REGION Network 25: PART A STATION 2 COLOR STATUS
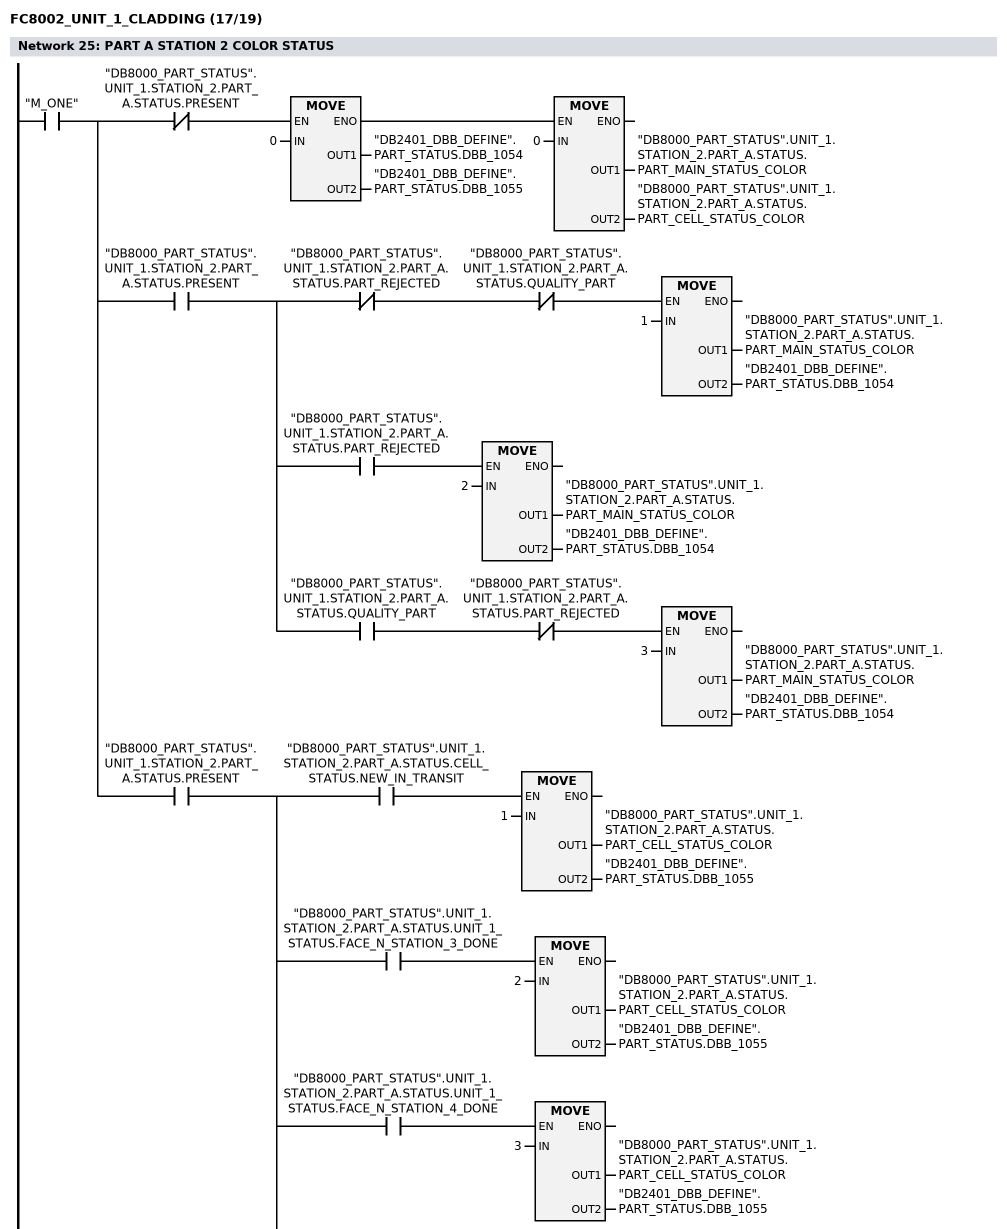
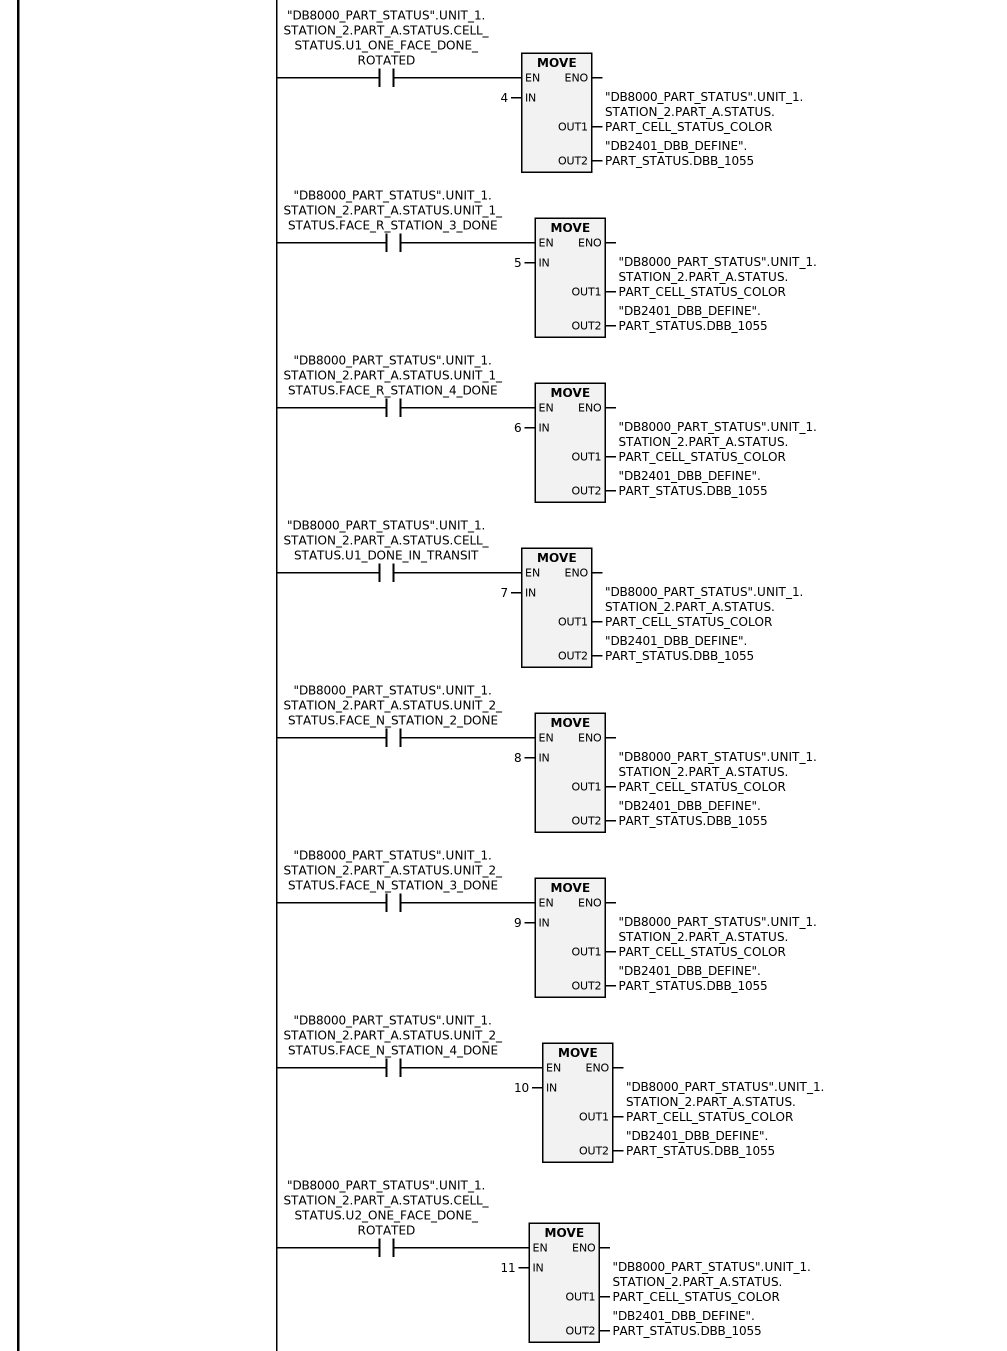
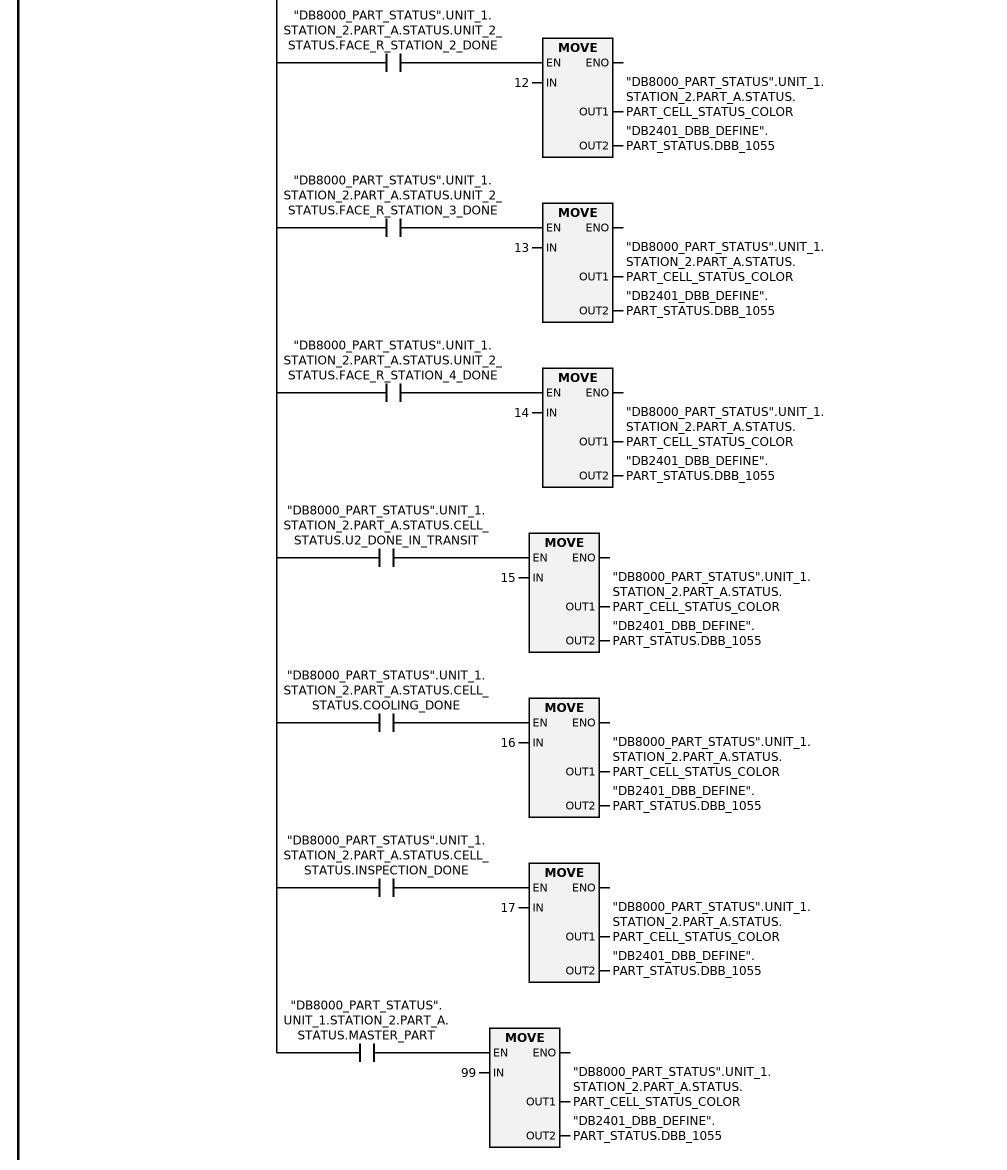
   RUNG wire#powerrail
      Contact( "M_ONE" )
      wire#w1
      I_Contact( "DB8000_PART_STATUS".UNIT_1.STATION_2.PART_A.STATUS.PRESENT )
      { S7_GenerateENO := "TRUE" } Move(in := 0, out1 => "DB2401_DBB_DEFINE".PART_STATUS.DBB_1054, out2 => "DB2401_DBB_DEFINE".PART_STATUS.DBB_1055)
      { S7_GenerateENO := "TRUE" } Move(in := 0, out1 => "DB8000_PART_STATUS".UNIT_1.STATION_2.PART_A.STATUS.PART_MAIN_STATUS_COLOR, out2 => "DB8000_PART_STATUS".UNIT_1.STATION_2.PART_A.STATUS.PART_CELL_STATUS_COLOR)
   END_RUNG
   RUNG wire#w1
      Contact( "DB8000_PART_STATUS".UNIT_1.STATION_2.PART_A.STATUS.PRESENT )
      wire#w2
      I_Contact( "DB8000_PART_STATUS".UNIT_1.STATION_2.PART_A.STATUS.PART_REJECTED )
      I_Contact( "DB8000_PART_STATUS".UNIT_1.STATION_2.PART_A.STATUS.QUALITY_PART )
      { S7_GenerateENO := "TRUE" } Move(in := 1, out1 => "DB8000_PART_STATUS".UNIT_1.STATION_2.PART_A.STATUS.PART_MAIN_STATUS_COLOR, out2 => "DB2401_DBB_DEFINE".PART_STATUS.DBB_1054)
   END_RUNG
   RUNG wire#w2
      Contact( "DB8000_PART_STATUS".UNIT_1.STATION_2.PART_A.STATUS.PART_REJECTED )
      { S7_GenerateENO := "TRUE" } Move(in := 2, out1 => "DB8000_PART_STATUS".UNIT_1.STATION_2.PART_A.STATUS.PART_MAIN_STATUS_COLOR, out2 => "DB2401_DBB_DEFINE".PART_STATUS.DBB_1054)
   END_RUNG
   RUNG wire#w2
      Contact( "DB8000_PART_STATUS".UNIT_1.STATION_2.PART_A.STATUS.QUALITY_PART )
      I_Contact( "DB8000_PART_STATUS".UNIT_1.STATION_2.PART_A.STATUS.PART_REJECTED )
      { S7_GenerateENO := "TRUE" } Move(in := 3, out1 => "DB8000_PART_STATUS".UNIT_1.STATION_2.PART_A.STATUS.PART_MAIN_STATUS_COLOR, out2 => "DB2401_DBB_DEFINE".PART_STATUS.DBB_1054)
   END_RUNG
   RUNG wire#w1
      Contact( "DB8000_PART_STATUS".UNIT_1.STATION_2.PART_A.STATUS.PRESENT )
      wire#w3
      Contact( "DB8000_PART_STATUS".UNIT_1.STATION_2.PART_A.STATUS.CELL_STATUS.NEW_IN_TRANSIT )
      { S7_GenerateENO := "TRUE" } Move(in := 1, out1 => "DB8000_PART_STATUS".UNIT_1.STATION_2.PART_A.STATUS.PART_CELL_STATUS_COLOR, out2 => "DB2401_DBB_DEFINE".PART_STATUS.DBB_1055)
   END_RUNG
   RUNG wire#w3
      Contact( "DB8000_PART_STATUS".UNIT_1.STATION_2.PART_A.STATUS.UNIT_1_STATUS.FACE_N_STATION_3_DONE )
      { S7_GenerateENO := "TRUE" } Move(in := 2, out1 => "DB8000_PART_STATUS".UNIT_1.STATION_2.PART_A.STATUS.PART_CELL_STATUS_COLOR, out2 => "DB2401_DBB_DEFINE".PART_STATUS.DBB_1055)
   END_RUNG
   RUNG wire#w3
      Contact( "DB8000_PART_STATUS".UNIT_1.STATION_2.PART_A.STATUS.UNIT_1_STATUS.FACE_N_STATION_4_DONE )
      { S7_GenerateENO := "TRUE" } Move(in := 3, out1 => "DB8000_PART_STATUS".UNIT_1.STATION_2.PART_A.STATUS.PART_CELL_STATUS_COLOR, out2 => "DB2401_DBB_DEFINE".PART_STATUS.DBB_1055)
   END_RUNG
   RUNG wire#w3
      Contact( "DB8000_PART_STATUS".UNIT_1.STATION_2.PART_A.STATUS.CELL_STATUS.U1_ONE_FACE_DONE_ROTATED )
      { S7_GenerateENO := "TRUE" } Move(in := 4, out1 => "DB8000_PART_STATUS".UNIT_1.STATION_2.PART_A.STATUS.PART_CELL_STATUS_COLOR, out2 => "DB2401_DBB_DEFINE".PART_STATUS.DBB_1055)
   END_RUNG
   RUNG wire#w3
      Contact( "DB8000_PART_STATUS".UNIT_1.STATION_2.PART_A.STATUS.UNIT_1_STATUS.FACE_R_STATION_3_DONE )
      { S7_GenerateENO := "TRUE" } Move(in := 5, out1 => "DB8000_PART_STATUS".UNIT_1.STATION_2.PART_A.STATUS.PART_CELL_STATUS_COLOR, out2 => "DB2401_DBB_DEFINE".PART_STATUS.DBB_1055)
   END_RUNG
   RUNG wire#w3
      Contact( "DB8000_PART_STATUS".UNIT_1.STATION_2.PART_A.STATUS.UNIT_1_STATUS.FACE_R_STATION_4_DONE )
      { S7_GenerateENO := "TRUE" } Move(in := 6, out1 => "DB8000_PART_STATUS".UNIT_1.STATION_2.PART_A.STATUS.PART_CELL_STATUS_COLOR, out2 => "DB2401_DBB_DEFINE".PART_STATUS.DBB_1055)
   END_RUNG
   RUNG wire#w3
      Contact( "DB8000_PART_STATUS".UNIT_1.STATION_2.PART_A.STATUS.CELL_STATUS.U1_DONE_IN_TRANSIT )
      { S7_GenerateENO := "TRUE" } Move(in := 7, out1 => "DB8000_PART_STATUS".UNIT_1.STATION_2.PART_A.STATUS.PART_CELL_STATUS_COLOR, out2 => "DB2401_DBB_DEFINE".PART_STATUS.DBB_1055)
   END_RUNG
   RUNG wire#w3
      Contact( "DB8000_PART_STATUS".UNIT_1.STATION_2.PART_A.STATUS.UNIT_2_STATUS.FACE_N_STATION_2_DONE )
      { S7_GenerateENO := "TRUE" } Move(in := 8, out1 => "DB8000_PART_STATUS".UNIT_1.STATION_2.PART_A.STATUS.PART_CELL_STATUS_COLOR, out2 => "DB2401_DBB_DEFINE".PART_STATUS.DBB_1055)
   END_RUNG
   RUNG wire#w3
      Contact( "DB8000_PART_STATUS".UNIT_1.STATION_2.PART_A.STATUS.UNIT_2_STATUS.FACE_N_STATION_3_DONE )
      Move(in := 9, out1 => "DB8000_PART_STATUS".UNIT_1.STATION_2.PART_A.STATUS.PART_CELL_STATUS_COLOR, out2 => "DB2401_DBB_DEFINE".PART_STATUS.DBB_1055)
   END_RUNG
   RUNG wire#w3
      Contact( "DB8000_PART_STATUS".UNIT_1.STATION_2.PART_A.STATUS.UNIT_2_STATUS.FACE_N_STATION_4_DONE )
      Move(in := 10, out1 => "DB8000_PART_STATUS".UNIT_1.STATION_2.PART_A.STATUS.PART_CELL_STATUS_COLOR, out2 => "DB2401_DBB_DEFINE".PART_STATUS.DBB_1055)
   END_RUNG
   RUNG wire#w3
      Contact( "DB8000_PART_STATUS".UNIT_1.STATION_2.PART_A.STATUS.CELL_STATUS.U2_ONE_FACE_DONE_ROTATED )
      Move(in := 11, out1 => "DB8000_PART_STATUS".UNIT_1.STATION_2.PART_A.STATUS.PART_CELL_STATUS_COLOR, out2 => "DB2401_DBB_DEFINE".PART_STATUS.DBB_1055)
   END_RUNG
   RUNG wire#w3
      Contact( "DB8000_PART_STATUS".UNIT_1.STATION_2.PART_A.STATUS.UNIT_2_STATUS.FACE_R_STATION_2_DONE )
      Move(in := 12, out1 => "DB8000_PART_STATUS".UNIT_1.STATION_2.PART_A.STATUS.PART_CELL_STATUS_COLOR, out2 => "DB2401_DBB_DEFINE".PART_STATUS.DBB_1055)
   END_RUNG
   RUNG wire#w3
      Contact( "DB8000_PART_STATUS".UNIT_1.STATION_2.PART_A.STATUS.UNIT_2_STATUS.FACE_R_STATION_3_DONE )
      Move(in := 13, out1 => "DB8000_PART_STATUS".UNIT_1.STATION_2.PART_A.STATUS.PART_CELL_STATUS_COLOR, out2 => "DB2401_DBB_DEFINE".PART_STATUS.DBB_1055)
   END_RUNG
   RUNG wire#w3
      Contact( "DB8000_PART_STATUS".UNIT_1.STATION_2.PART_A.STATUS.UNIT_2_STATUS.FACE_R_STATION_4_DONE )
      Move(in := 14, out1 => "DB8000_PART_STATUS".UNIT_1.STATION_2.PART_A.STATUS.PART_CELL_STATUS_COLOR, out2 => "DB2401_DBB_DEFINE".PART_STATUS.DBB_1055)
   END_RUNG
   RUNG wire#w3
      Contact( "DB8000_PART_STATUS".UNIT_1.STATION_2.PART_A.STATUS.CELL_STATUS.U2_DONE_IN_TRANSIT )
      Move(in := 15, out1 => "DB8000_PART_STATUS".UNIT_1.STATION_2.PART_A.STATUS.PART_CELL_STATUS_COLOR, out2 => "DB2401_DBB_DEFINE".PART_STATUS.DBB_1055)
   END_RUNG
   RUNG wire#w3
      Contact( "DB8000_PART_STATUS".UNIT_1.STATION_2.PART_A.STATUS.CELL_STATUS.COOLING_DONE )
      Move(in := 16, out1 => "DB8000_PART_STATUS".UNIT_1.STATION_2.PART_A.STATUS.PART_CELL_STATUS_COLOR, out2 => "DB2401_DBB_DEFINE".PART_STATUS.DBB_1055)
   END_RUNG
   RUNG wire#w3
      Contact( "DB8000_PART_STATUS".UNIT_1.STATION_2.PART_A.STATUS.CELL_STATUS.INSPECTION_DONE )
      Move(in := 17, out1 => "DB8000_PART_STATUS".UNIT_1.STATION_2.PART_A.STATUS.PART_CELL_STATUS_COLOR, out2 => "DB2401_DBB_DEFINE".PART_STATUS.DBB_1055)
   END_RUNG
   RUNG wire#w3
      Contact( "DB8000_PART_STATUS".UNIT_1.STATION_2.PART_A.STATUS.MASTER_PART )
      Move(in := 99, out1 => "DB8000_PART_STATUS".UNIT_1.STATION_2.PART_A.STATUS.PART_CELL_STATUS_COLOR, out2 => "DB2401_DBB_DEFINE".PART_STATUS.DBB_1055)
   END_RUNG
   // the same network as SCL:
   // ENO of a box is taken as its EN; it also drops when the box reports an error
   IF "M_ONE" AND NOT "DB8000_PART_STATUS".UNIT_1.STATION_2.PART_A.STATUS.PRESENT THEN
       "DB2401_DBB_DEFINE".PART_STATUS.DBB_1054 := 0;
       "DB2401_DBB_DEFINE".PART_STATUS.DBB_1055 := 0;
       "DB8000_PART_STATUS".UNIT_1.STATION_2.PART_A.STATUS.PART_MAIN_STATUS_COLOR := 0;
       "DB8000_PART_STATUS".UNIT_1.STATION_2.PART_A.STATUS.PART_CELL_STATUS_COLOR := 0;
   END_IF;
   #_w1 := "M_ONE" AND "DB8000_PART_STATUS".UNIT_1.STATION_2.PART_A.STATUS.PRESENT;
   IF #_w1 AND NOT "DB8000_PART_STATUS".UNIT_1.STATION_2.PART_A.STATUS.PART_REJECTED AND NOT "DB8000_PART_STATUS".UNIT_1.STATION_2.PART_A.STATUS.QUALITY_PART THEN
       "DB8000_PART_STATUS".UNIT_1.STATION_2.PART_A.STATUS.PART_MAIN_STATUS_COLOR := 1;
       "DB2401_DBB_DEFINE".PART_STATUS.DBB_1054 := 1;
   END_IF;
   IF #_w1 AND "DB8000_PART_STATUS".UNIT_1.STATION_2.PART_A.STATUS.PART_REJECTED THEN
       "DB8000_PART_STATUS".UNIT_1.STATION_2.PART_A.STATUS.PART_MAIN_STATUS_COLOR := 2;
       "DB2401_DBB_DEFINE".PART_STATUS.DBB_1054 := 2;
   END_IF;
   IF #_w1 AND "DB8000_PART_STATUS".UNIT_1.STATION_2.PART_A.STATUS.QUALITY_PART AND NOT "DB8000_PART_STATUS".UNIT_1.STATION_2.PART_A.STATUS.PART_REJECTED THEN
       "DB8000_PART_STATUS".UNIT_1.STATION_2.PART_A.STATUS.PART_MAIN_STATUS_COLOR := 3;
       "DB2401_DBB_DEFINE".PART_STATUS.DBB_1054 := 3;
   END_IF;
   #_w2 := "M_ONE" AND "DB8000_PART_STATUS".UNIT_1.STATION_2.PART_A.STATUS.PRESENT;
   IF #_w2 AND "DB8000_PART_STATUS".UNIT_1.STATION_2.PART_A.STATUS.CELL_STATUS.NEW_IN_TRANSIT THEN
       "DB8000_PART_STATUS".UNIT_1.STATION_2.PART_A.STATUS.PART_CELL_STATUS_COLOR := 1;
       "DB2401_DBB_DEFINE".PART_STATUS.DBB_1055 := 1;
   END_IF;
   IF #_w2 AND "DB8000_PART_STATUS".UNIT_1.STATION_2.PART_A.STATUS.UNIT_1_STATUS.FACE_N_STATION_3_DONE THEN
       "DB8000_PART_STATUS".UNIT_1.STATION_2.PART_A.STATUS.PART_CELL_STATUS_COLOR := 2;
       "DB2401_DBB_DEFINE".PART_STATUS.DBB_1055 := 2;
   END_IF;
   IF #_w2 AND "DB8000_PART_STATUS".UNIT_1.STATION_2.PART_A.STATUS.UNIT_1_STATUS.FACE_N_STATION_4_DONE THEN
       "DB8000_PART_STATUS".UNIT_1.STATION_2.PART_A.STATUS.PART_CELL_STATUS_COLOR := 3;
       "DB2401_DBB_DEFINE".PART_STATUS.DBB_1055 := 3;
   END_IF;
   IF #_w2 AND "DB8000_PART_STATUS".UNIT_1.STATION_2.PART_A.STATUS.CELL_STATUS.U1_ONE_FACE_DONE_ROTATED THEN
       "DB8000_PART_STATUS".UNIT_1.STATION_2.PART_A.STATUS.PART_CELL_STATUS_COLOR := 4;
       "DB2401_DBB_DEFINE".PART_STATUS.DBB_1055 := 4;
   END_IF;
   IF #_w2 AND "DB8000_PART_STATUS".UNIT_1.STATION_2.PART_A.STATUS.UNIT_1_STATUS.FACE_R_STATION_3_DONE THEN
       "DB8000_PART_STATUS".UNIT_1.STATION_2.PART_A.STATUS.PART_CELL_STATUS_COLOR := 5;
       "DB2401_DBB_DEFINE".PART_STATUS.DBB_1055 := 5;
   END_IF;
   IF #_w2 AND "DB8000_PART_STATUS".UNIT_1.STATION_2.PART_A.STATUS.UNIT_1_STATUS.FACE_R_STATION_4_DONE THEN
       "DB8000_PART_STATUS".UNIT_1.STATION_2.PART_A.STATUS.PART_CELL_STATUS_COLOR := 6;
       "DB2401_DBB_DEFINE".PART_STATUS.DBB_1055 := 6;
   END_IF;
   IF #_w2 AND "DB8000_PART_STATUS".UNIT_1.STATION_2.PART_A.STATUS.CELL_STATUS.U1_DONE_IN_TRANSIT THEN
       "DB8000_PART_STATUS".UNIT_1.STATION_2.PART_A.STATUS.PART_CELL_STATUS_COLOR := 7;
       "DB2401_DBB_DEFINE".PART_STATUS.DBB_1055 := 7;
   END_IF;
   IF #_w2 AND "DB8000_PART_STATUS".UNIT_1.STATION_2.PART_A.STATUS.UNIT_2_STATUS.FACE_N_STATION_2_DONE THEN
       "DB8000_PART_STATUS".UNIT_1.STATION_2.PART_A.STATUS.PART_CELL_STATUS_COLOR := 8;
       "DB2401_DBB_DEFINE".PART_STATUS.DBB_1055 := 8;
   END_IF;
   IF #_w2 AND "DB8000_PART_STATUS".UNIT_1.STATION_2.PART_A.STATUS.UNIT_2_STATUS.FACE_N_STATION_3_DONE THEN
       "DB8000_PART_STATUS".UNIT_1.STATION_2.PART_A.STATUS.PART_CELL_STATUS_COLOR := 9;
       "DB2401_DBB_DEFINE".PART_STATUS.DBB_1055 := 9;
   END_IF;
   IF #_w2 AND "DB8000_PART_STATUS".UNIT_1.STATION_2.PART_A.STATUS.UNIT_2_STATUS.FACE_N_STATION_4_DONE THEN
       "DB8000_PART_STATUS".UNIT_1.STATION_2.PART_A.STATUS.PART_CELL_STATUS_COLOR := 10;
       "DB2401_DBB_DEFINE".PART_STATUS.DBB_1055 := 10;
   END_IF;
   IF #_w2 AND "DB8000_PART_STATUS".UNIT_1.STATION_2.PART_A.STATUS.CELL_STATUS.U2_ONE_FACE_DONE_ROTATED THEN
       "DB8000_PART_STATUS".UNIT_1.STATION_2.PART_A.STATUS.PART_CELL_STATUS_COLOR := 11;
       "DB2401_DBB_DEFINE".PART_STATUS.DBB_1055 := 11;
   END_IF;
   IF #_w2 AND "DB8000_PART_STATUS".UNIT_1.STATION_2.PART_A.STATUS.UNIT_2_STATUS.FACE_R_STATION_2_DONE THEN
       "DB8000_PART_STATUS".UNIT_1.STATION_2.PART_A.STATUS.PART_CELL_STATUS_COLOR := 12;
       "DB2401_DBB_DEFINE".PART_STATUS.DBB_1055 := 12;
   END_IF;
   IF #_w2 AND "DB8000_PART_STATUS".UNIT_1.STATION_2.PART_A.STATUS.UNIT_2_STATUS.FACE_R_STATION_3_DONE THEN
       "DB8000_PART_STATUS".UNIT_1.STATION_2.PART_A.STATUS.PART_CELL_STATUS_COLOR := 13;
       "DB2401_DBB_DEFINE".PART_STATUS.DBB_1055 := 13;
   END_IF;
   IF #_w2 AND "DB8000_PART_STATUS".UNIT_1.STATION_2.PART_A.STATUS.UNIT_2_STATUS.FACE_R_STATION_4_DONE THEN
       "DB8000_PART_STATUS".UNIT_1.STATION_2.PART_A.STATUS.PART_CELL_STATUS_COLOR := 14;
       "DB2401_DBB_DEFINE".PART_STATUS.DBB_1055 := 14;
   END_IF;
   IF #_w2 AND "DB8000_PART_STATUS".UNIT_1.STATION_2.PART_A.STATUS.CELL_STATUS.U2_DONE_IN_TRANSIT THEN
       "DB8000_PART_STATUS".UNIT_1.STATION_2.PART_A.STATUS.PART_CELL_STATUS_COLOR := 15;
       "DB2401_DBB_DEFINE".PART_STATUS.DBB_1055 := 15;
   END_IF;
   IF #_w2 AND "DB8000_PART_STATUS".UNIT_1.STATION_2.PART_A.STATUS.CELL_STATUS.COOLING_DONE THEN
       "DB8000_PART_STATUS".UNIT_1.STATION_2.PART_A.STATUS.PART_CELL_STATUS_COLOR := 16;
       "DB2401_DBB_DEFINE".PART_STATUS.DBB_1055 := 16;
   END_IF;
   IF #_w2 AND "DB8000_PART_STATUS".UNIT_1.STATION_2.PART_A.STATUS.CELL_STATUS.INSPECTION_DONE THEN
       "DB8000_PART_STATUS".UNIT_1.STATION_2.PART_A.STATUS.PART_CELL_STATUS_COLOR := 17;
       "DB2401_DBB_DEFINE".PART_STATUS.DBB_1055 := 17;
   END_IF;
   IF #_w2 AND "DB8000_PART_STATUS".UNIT_1.STATION_2.PART_A.STATUS.MASTER_PART THEN
       "DB8000_PART_STATUS".UNIT_1.STATION_2.PART_A.STATUS.PART_CELL_STATUS_COLOR := 99;
       "DB2401_DBB_DEFINE".PART_STATUS.DBB_1055 := 99;
   END_IF;
END_REGION

REGION Network 26: PART A STATION 3 COLOR STATUS
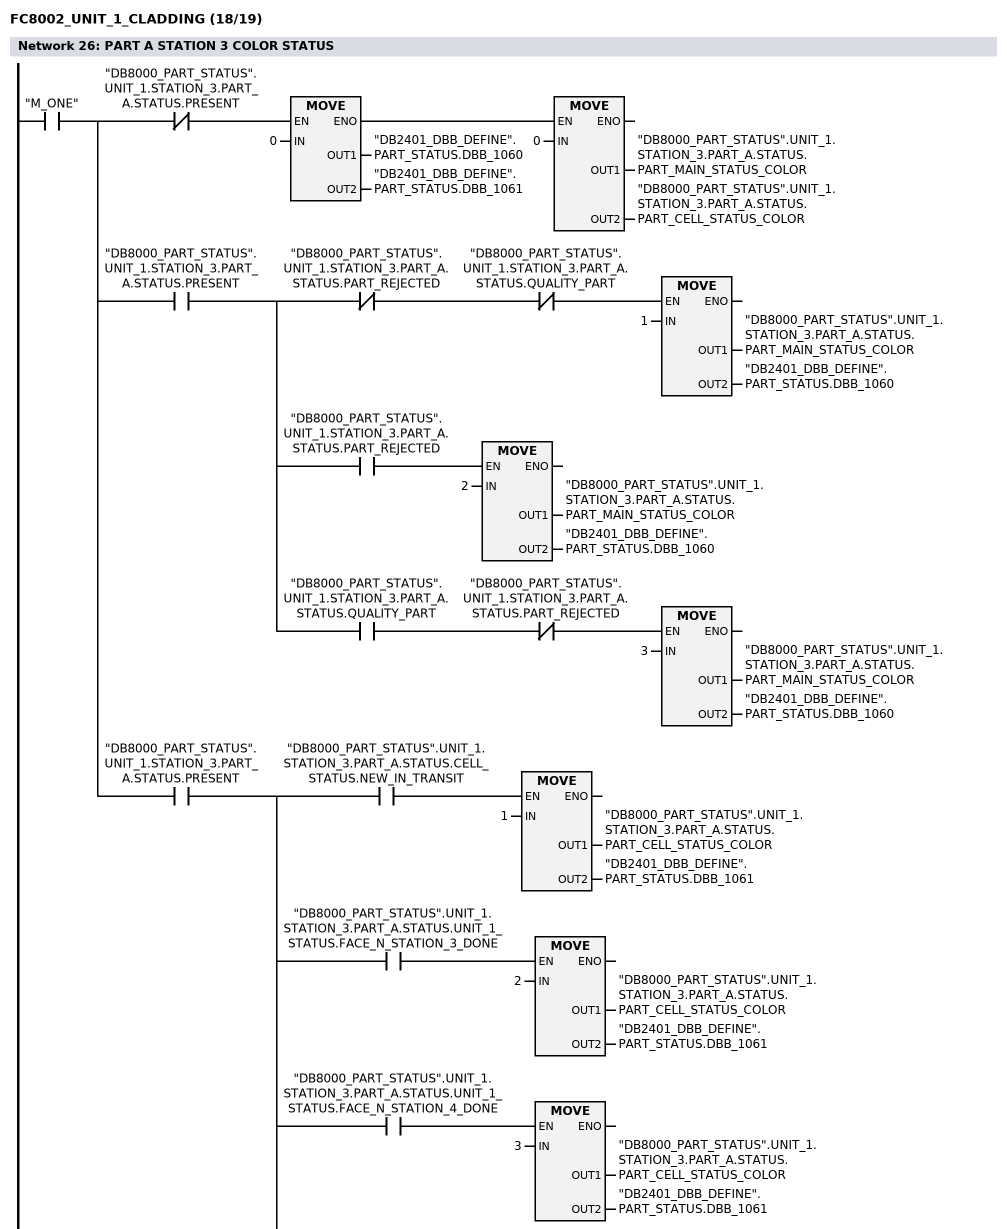
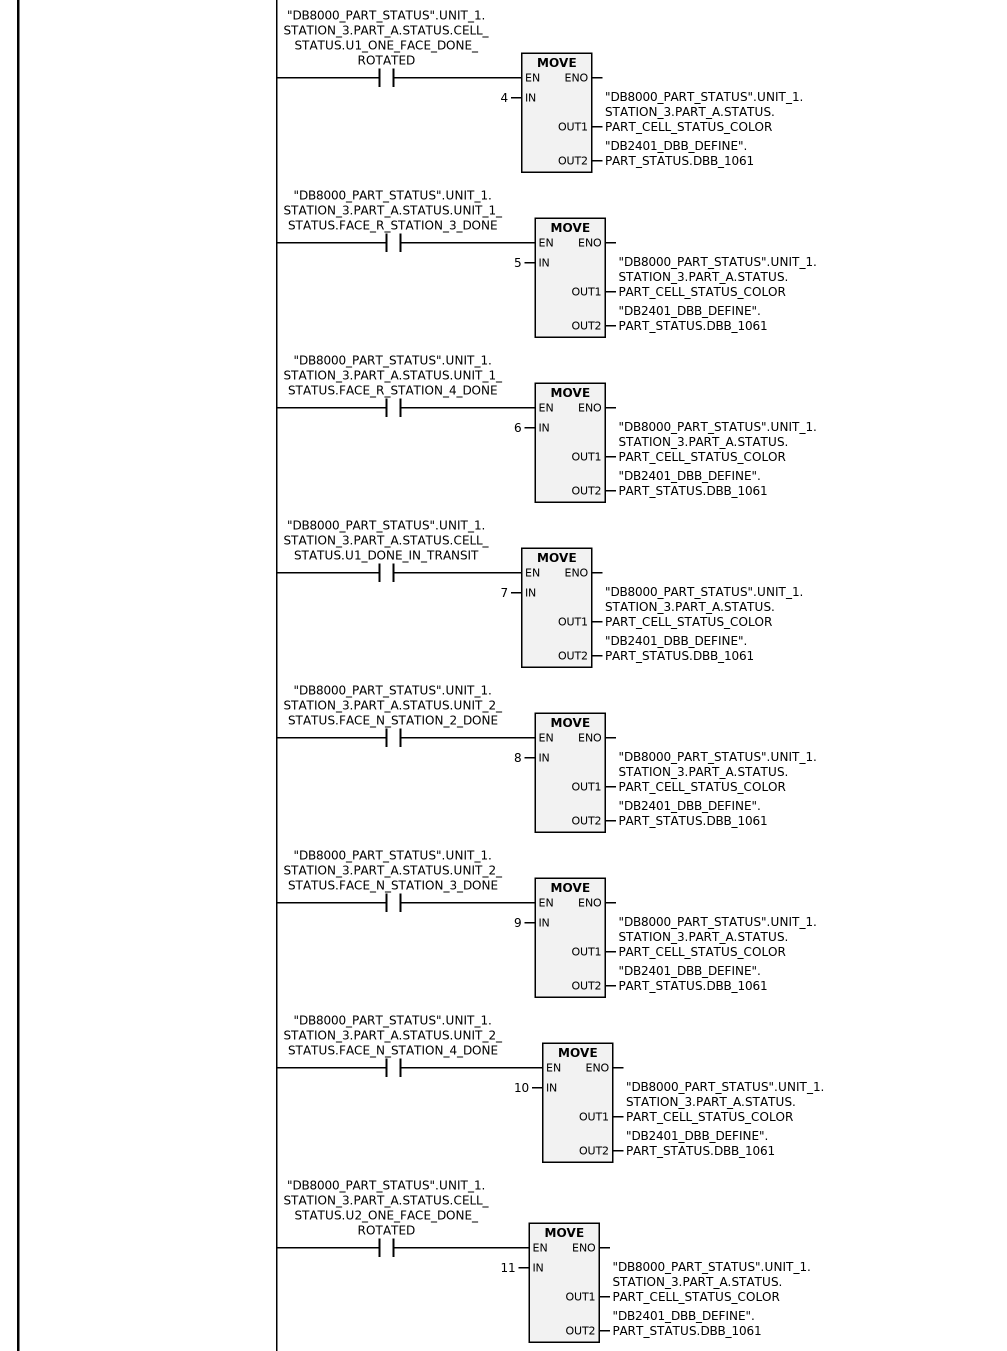
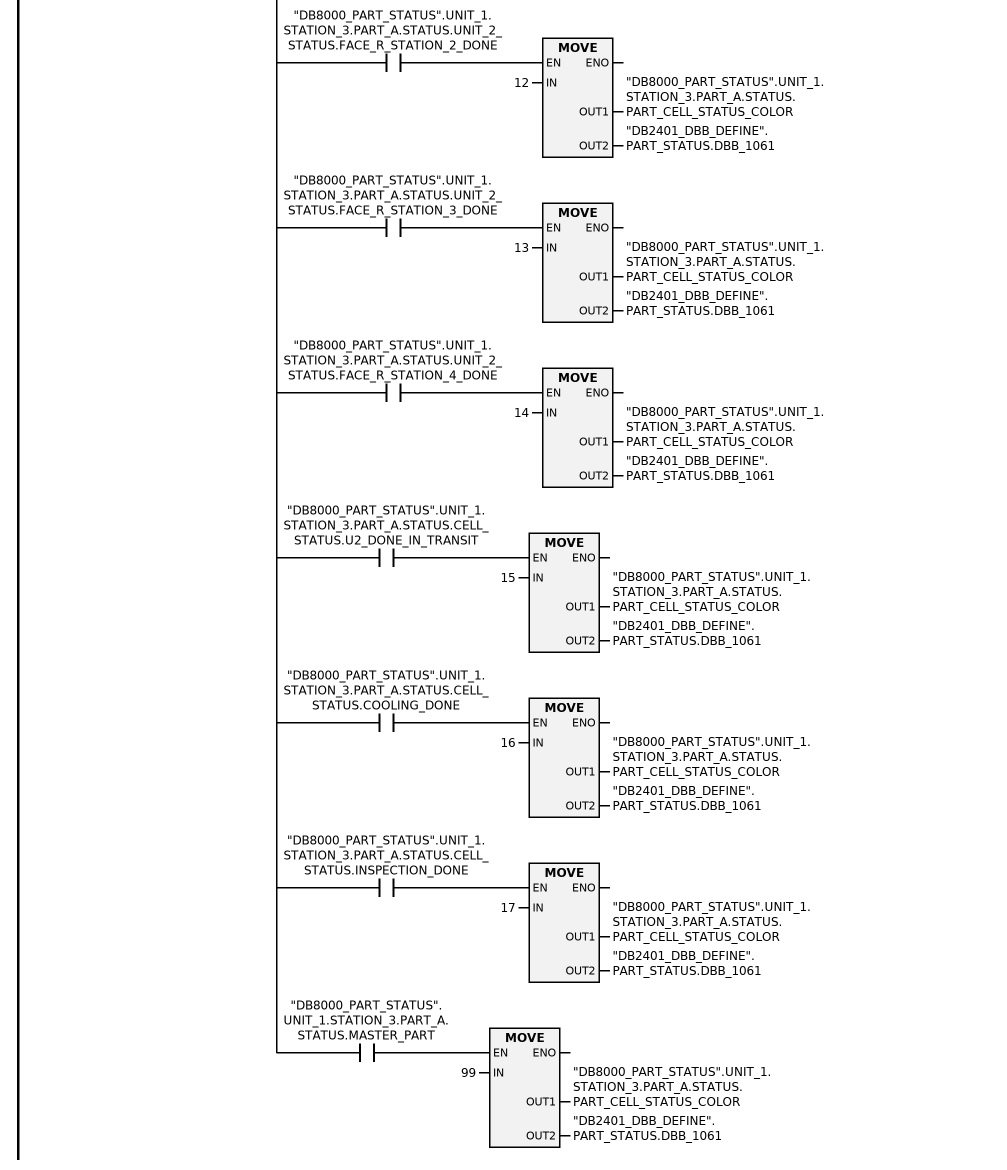
   RUNG wire#powerrail
      Contact( "M_ONE" )
      wire#w1
      I_Contact( "DB8000_PART_STATUS".UNIT_1.STATION_3.PART_A.STATUS.PRESENT )
      { S7_GenerateENO := "TRUE" } Move(in := 0, out1 => "DB2401_DBB_DEFINE".PART_STATUS.DBB_1060, out2 => "DB2401_DBB_DEFINE".PART_STATUS.DBB_1061)
      { S7_GenerateENO := "TRUE" } Move(in := 0, out1 => "DB8000_PART_STATUS".UNIT_1.STATION_3.PART_A.STATUS.PART_MAIN_STATUS_COLOR, out2 => "DB8000_PART_STATUS".UNIT_1.STATION_3.PART_A.STATUS.PART_CELL_STATUS_COLOR)
   END_RUNG
   RUNG wire#w1
      Contact( "DB8000_PART_STATUS".UNIT_1.STATION_3.PART_A.STATUS.PRESENT )
      wire#w2
      I_Contact( "DB8000_PART_STATUS".UNIT_1.STATION_3.PART_A.STATUS.PART_REJECTED )
      I_Contact( "DB8000_PART_STATUS".UNIT_1.STATION_3.PART_A.STATUS.QUALITY_PART )
      { S7_GenerateENO := "TRUE" } Move(in := 1, out1 => "DB8000_PART_STATUS".UNIT_1.STATION_3.PART_A.STATUS.PART_MAIN_STATUS_COLOR, out2 => "DB2401_DBB_DEFINE".PART_STATUS.DBB_1060)
   END_RUNG
   RUNG wire#w2
      Contact( "DB8000_PART_STATUS".UNIT_1.STATION_3.PART_A.STATUS.PART_REJECTED )
      { S7_GenerateENO := "TRUE" } Move(in := 2, out1 => "DB8000_PART_STATUS".UNIT_1.STATION_3.PART_A.STATUS.PART_MAIN_STATUS_COLOR, out2 => "DB2401_DBB_DEFINE".PART_STATUS.DBB_1060)
   END_RUNG
   RUNG wire#w2
      Contact( "DB8000_PART_STATUS".UNIT_1.STATION_3.PART_A.STATUS.QUALITY_PART )
      I_Contact( "DB8000_PART_STATUS".UNIT_1.STATION_3.PART_A.STATUS.PART_REJECTED )
      { S7_GenerateENO := "TRUE" } Move(in := 3, out1 => "DB8000_PART_STATUS".UNIT_1.STATION_3.PART_A.STATUS.PART_MAIN_STATUS_COLOR, out2 => "DB2401_DBB_DEFINE".PART_STATUS.DBB_1060)
   END_RUNG
   RUNG wire#w1
      Contact( "DB8000_PART_STATUS".UNIT_1.STATION_3.PART_A.STATUS.PRESENT )
      wire#w3
      Contact( "DB8000_PART_STATUS".UNIT_1.STATION_3.PART_A.STATUS.CELL_STATUS.NEW_IN_TRANSIT )
      { S7_GenerateENO := "TRUE" } Move(in := 1, out1 => "DB8000_PART_STATUS".UNIT_1.STATION_3.PART_A.STATUS.PART_CELL_STATUS_COLOR, out2 => "DB2401_DBB_DEFINE".PART_STATUS.DBB_1061)
   END_RUNG
   RUNG wire#w3
      Contact( "DB8000_PART_STATUS".UNIT_1.STATION_3.PART_A.STATUS.UNIT_1_STATUS.FACE_N_STATION_3_DONE )
      { S7_GenerateENO := "TRUE" } Move(in := 2, out1 => "DB8000_PART_STATUS".UNIT_1.STATION_3.PART_A.STATUS.PART_CELL_STATUS_COLOR, out2 => "DB2401_DBB_DEFINE".PART_STATUS.DBB_1061)
   END_RUNG
   RUNG wire#w3
      Contact( "DB8000_PART_STATUS".UNIT_1.STATION_3.PART_A.STATUS.UNIT_1_STATUS.FACE_N_STATION_4_DONE )
      { S7_GenerateENO := "TRUE" } Move(in := 3, out1 => "DB8000_PART_STATUS".UNIT_1.STATION_3.PART_A.STATUS.PART_CELL_STATUS_COLOR, out2 => "DB2401_DBB_DEFINE".PART_STATUS.DBB_1061)
   END_RUNG
   RUNG wire#w3
      Contact( "DB8000_PART_STATUS".UNIT_1.STATION_3.PART_A.STATUS.CELL_STATUS.U1_ONE_FACE_DONE_ROTATED )
      { S7_GenerateENO := "TRUE" } Move(in := 4, out1 => "DB8000_PART_STATUS".UNIT_1.STATION_3.PART_A.STATUS.PART_CELL_STATUS_COLOR, out2 => "DB2401_DBB_DEFINE".PART_STATUS.DBB_1061)
   END_RUNG
   RUNG wire#w3
      Contact( "DB8000_PART_STATUS".UNIT_1.STATION_3.PART_A.STATUS.UNIT_1_STATUS.FACE_R_STATION_3_DONE )
      { S7_GenerateENO := "TRUE" } Move(in := 5, out1 => "DB8000_PART_STATUS".UNIT_1.STATION_3.PART_A.STATUS.PART_CELL_STATUS_COLOR, out2 => "DB2401_DBB_DEFINE".PART_STATUS.DBB_1061)
   END_RUNG
   RUNG wire#w3
      Contact( "DB8000_PART_STATUS".UNIT_1.STATION_3.PART_A.STATUS.UNIT_1_STATUS.FACE_R_STATION_4_DONE )
      { S7_GenerateENO := "TRUE" } Move(in := 6, out1 => "DB8000_PART_STATUS".UNIT_1.STATION_3.PART_A.STATUS.PART_CELL_STATUS_COLOR, out2 => "DB2401_DBB_DEFINE".PART_STATUS.DBB_1061)
   END_RUNG
   RUNG wire#w3
      Contact( "DB8000_PART_STATUS".UNIT_1.STATION_3.PART_A.STATUS.CELL_STATUS.U1_DONE_IN_TRANSIT )
      { S7_GenerateENO := "TRUE" } Move(in := 7, out1 => "DB8000_PART_STATUS".UNIT_1.STATION_3.PART_A.STATUS.PART_CELL_STATUS_COLOR, out2 => "DB2401_DBB_DEFINE".PART_STATUS.DBB_1061)
   END_RUNG
   RUNG wire#w3
      Contact( "DB8000_PART_STATUS".UNIT_1.STATION_3.PART_A.STATUS.UNIT_2_STATUS.FACE_N_STATION_2_DONE )
      { S7_GenerateENO := "TRUE" } Move(in := 8, out1 => "DB8000_PART_STATUS".UNIT_1.STATION_3.PART_A.STATUS.PART_CELL_STATUS_COLOR, out2 => "DB2401_DBB_DEFINE".PART_STATUS.DBB_1061)
   END_RUNG
   RUNG wire#w3
      Contact( "DB8000_PART_STATUS".UNIT_1.STATION_3.PART_A.STATUS.UNIT_2_STATUS.FACE_N_STATION_3_DONE )
      Move(in := 9, out1 => "DB8000_PART_STATUS".UNIT_1.STATION_3.PART_A.STATUS.PART_CELL_STATUS_COLOR, out2 => "DB2401_DBB_DEFINE".PART_STATUS.DBB_1061)
   END_RUNG
   RUNG wire#w3
      Contact( "DB8000_PART_STATUS".UNIT_1.STATION_3.PART_A.STATUS.UNIT_2_STATUS.FACE_N_STATION_4_DONE )
      Move(in := 10, out1 => "DB8000_PART_STATUS".UNIT_1.STATION_3.PART_A.STATUS.PART_CELL_STATUS_COLOR, out2 => "DB2401_DBB_DEFINE".PART_STATUS.DBB_1061)
   END_RUNG
   RUNG wire#w3
      Contact( "DB8000_PART_STATUS".UNIT_1.STATION_3.PART_A.STATUS.CELL_STATUS.U2_ONE_FACE_DONE_ROTATED )
      Move(in := 11, out1 => "DB8000_PART_STATUS".UNIT_1.STATION_3.PART_A.STATUS.PART_CELL_STATUS_COLOR, out2 => "DB2401_DBB_DEFINE".PART_STATUS.DBB_1061)
   END_RUNG
   RUNG wire#w3
      Contact( "DB8000_PART_STATUS".UNIT_1.STATION_3.PART_A.STATUS.UNIT_2_STATUS.FACE_R_STATION_2_DONE )
      Move(in := 12, out1 => "DB8000_PART_STATUS".UNIT_1.STATION_3.PART_A.STATUS.PART_CELL_STATUS_COLOR, out2 => "DB2401_DBB_DEFINE".PART_STATUS.DBB_1061)
   END_RUNG
   RUNG wire#w3
      Contact( "DB8000_PART_STATUS".UNIT_1.STATION_3.PART_A.STATUS.UNIT_2_STATUS.FACE_R_STATION_3_DONE )
      Move(in := 13, out1 => "DB8000_PART_STATUS".UNIT_1.STATION_3.PART_A.STATUS.PART_CELL_STATUS_COLOR, out2 => "DB2401_DBB_DEFINE".PART_STATUS.DBB_1061)
   END_RUNG
   RUNG wire#w3
      Contact( "DB8000_PART_STATUS".UNIT_1.STATION_3.PART_A.STATUS.UNIT_2_STATUS.FACE_R_STATION_4_DONE )
      Move(in := 14, out1 => "DB8000_PART_STATUS".UNIT_1.STATION_3.PART_A.STATUS.PART_CELL_STATUS_COLOR, out2 => "DB2401_DBB_DEFINE".PART_STATUS.DBB_1061)
   END_RUNG
   RUNG wire#w3
      Contact( "DB8000_PART_STATUS".UNIT_1.STATION_3.PART_A.STATUS.CELL_STATUS.U2_DONE_IN_TRANSIT )
      Move(in := 15, out1 => "DB8000_PART_STATUS".UNIT_1.STATION_3.PART_A.STATUS.PART_CELL_STATUS_COLOR, out2 => "DB2401_DBB_DEFINE".PART_STATUS.DBB_1061)
   END_RUNG
   RUNG wire#w3
      Contact( "DB8000_PART_STATUS".UNIT_1.STATION_3.PART_A.STATUS.CELL_STATUS.COOLING_DONE )
      Move(in := 16, out1 => "DB8000_PART_STATUS".UNIT_1.STATION_3.PART_A.STATUS.PART_CELL_STATUS_COLOR, out2 => "DB2401_DBB_DEFINE".PART_STATUS.DBB_1061)
   END_RUNG
   RUNG wire#w3
      Contact( "DB8000_PART_STATUS".UNIT_1.STATION_3.PART_A.STATUS.CELL_STATUS.INSPECTION_DONE )
      Move(in := 17, out1 => "DB8000_PART_STATUS".UNIT_1.STATION_3.PART_A.STATUS.PART_CELL_STATUS_COLOR, out2 => "DB2401_DBB_DEFINE".PART_STATUS.DBB_1061)
   END_RUNG
   RUNG wire#w3
      Contact( "DB8000_PART_STATUS".UNIT_1.STATION_3.PART_A.STATUS.MASTER_PART )
      Move(in := 99, out1 => "DB8000_PART_STATUS".UNIT_1.STATION_3.PART_A.STATUS.PART_CELL_STATUS_COLOR, out2 => "DB2401_DBB_DEFINE".PART_STATUS.DBB_1061)
   END_RUNG
   // the same network as SCL:
   // ENO of a box is taken as its EN; it also drops when the box reports an error
   IF "M_ONE" AND NOT "DB8000_PART_STATUS".UNIT_1.STATION_3.PART_A.STATUS.PRESENT THEN
       "DB2401_DBB_DEFINE".PART_STATUS.DBB_1060 := 0;
       "DB2401_DBB_DEFINE".PART_STATUS.DBB_1061 := 0;
       "DB8000_PART_STATUS".UNIT_1.STATION_3.PART_A.STATUS.PART_MAIN_STATUS_COLOR := 0;
       "DB8000_PART_STATUS".UNIT_1.STATION_3.PART_A.STATUS.PART_CELL_STATUS_COLOR := 0;
   END_IF;
   #_w1 := "M_ONE" AND "DB8000_PART_STATUS".UNIT_1.STATION_3.PART_A.STATUS.PRESENT;
   IF #_w1 AND NOT "DB8000_PART_STATUS".UNIT_1.STATION_3.PART_A.STATUS.PART_REJECTED AND NOT "DB8000_PART_STATUS".UNIT_1.STATION_3.PART_A.STATUS.QUALITY_PART THEN
       "DB8000_PART_STATUS".UNIT_1.STATION_3.PART_A.STATUS.PART_MAIN_STATUS_COLOR := 1;
       "DB2401_DBB_DEFINE".PART_STATUS.DBB_1060 := 1;
   END_IF;
   IF #_w1 AND "DB8000_PART_STATUS".UNIT_1.STATION_3.PART_A.STATUS.PART_REJECTED THEN
       "DB8000_PART_STATUS".UNIT_1.STATION_3.PART_A.STATUS.PART_MAIN_STATUS_COLOR := 2;
       "DB2401_DBB_DEFINE".PART_STATUS.DBB_1060 := 2;
   END_IF;
   IF #_w1 AND "DB8000_PART_STATUS".UNIT_1.STATION_3.PART_A.STATUS.QUALITY_PART AND NOT "DB8000_PART_STATUS".UNIT_1.STATION_3.PART_A.STATUS.PART_REJECTED THEN
       "DB8000_PART_STATUS".UNIT_1.STATION_3.PART_A.STATUS.PART_MAIN_STATUS_COLOR := 3;
       "DB2401_DBB_DEFINE".PART_STATUS.DBB_1060 := 3;
   END_IF;
   #_w2 := "M_ONE" AND "DB8000_PART_STATUS".UNIT_1.STATION_3.PART_A.STATUS.PRESENT;
   IF #_w2 AND "DB8000_PART_STATUS".UNIT_1.STATION_3.PART_A.STATUS.CELL_STATUS.NEW_IN_TRANSIT THEN
       "DB8000_PART_STATUS".UNIT_1.STATION_3.PART_A.STATUS.PART_CELL_STATUS_COLOR := 1;
       "DB2401_DBB_DEFINE".PART_STATUS.DBB_1061 := 1;
   END_IF;
   IF #_w2 AND "DB8000_PART_STATUS".UNIT_1.STATION_3.PART_A.STATUS.UNIT_1_STATUS.FACE_N_STATION_3_DONE THEN
       "DB8000_PART_STATUS".UNIT_1.STATION_3.PART_A.STATUS.PART_CELL_STATUS_COLOR := 2;
       "DB2401_DBB_DEFINE".PART_STATUS.DBB_1061 := 2;
   END_IF;
   IF #_w2 AND "DB8000_PART_STATUS".UNIT_1.STATION_3.PART_A.STATUS.UNIT_1_STATUS.FACE_N_STATION_4_DONE THEN
       "DB8000_PART_STATUS".UNIT_1.STATION_3.PART_A.STATUS.PART_CELL_STATUS_COLOR := 3;
       "DB2401_DBB_DEFINE".PART_STATUS.DBB_1061 := 3;
   END_IF;
   IF #_w2 AND "DB8000_PART_STATUS".UNIT_1.STATION_3.PART_A.STATUS.CELL_STATUS.U1_ONE_FACE_DONE_ROTATED THEN
       "DB8000_PART_STATUS".UNIT_1.STATION_3.PART_A.STATUS.PART_CELL_STATUS_COLOR := 4;
       "DB2401_DBB_DEFINE".PART_STATUS.DBB_1061 := 4;
   END_IF;
   IF #_w2 AND "DB8000_PART_STATUS".UNIT_1.STATION_3.PART_A.STATUS.UNIT_1_STATUS.FACE_R_STATION_3_DONE THEN
       "DB8000_PART_STATUS".UNIT_1.STATION_3.PART_A.STATUS.PART_CELL_STATUS_COLOR := 5;
       "DB2401_DBB_DEFINE".PART_STATUS.DBB_1061 := 5;
   END_IF;
   IF #_w2 AND "DB8000_PART_STATUS".UNIT_1.STATION_3.PART_A.STATUS.UNIT_1_STATUS.FACE_R_STATION_4_DONE THEN
       "DB8000_PART_STATUS".UNIT_1.STATION_3.PART_A.STATUS.PART_CELL_STATUS_COLOR := 6;
       "DB2401_DBB_DEFINE".PART_STATUS.DBB_1061 := 6;
   END_IF;
   IF #_w2 AND "DB8000_PART_STATUS".UNIT_1.STATION_3.PART_A.STATUS.CELL_STATUS.U1_DONE_IN_TRANSIT THEN
       "DB8000_PART_STATUS".UNIT_1.STATION_3.PART_A.STATUS.PART_CELL_STATUS_COLOR := 7;
       "DB2401_DBB_DEFINE".PART_STATUS.DBB_1061 := 7;
   END_IF;
   IF #_w2 AND "DB8000_PART_STATUS".UNIT_1.STATION_3.PART_A.STATUS.UNIT_2_STATUS.FACE_N_STATION_2_DONE THEN
       "DB8000_PART_STATUS".UNIT_1.STATION_3.PART_A.STATUS.PART_CELL_STATUS_COLOR := 8;
       "DB2401_DBB_DEFINE".PART_STATUS.DBB_1061 := 8;
   END_IF;
   IF #_w2 AND "DB8000_PART_STATUS".UNIT_1.STATION_3.PART_A.STATUS.UNIT_2_STATUS.FACE_N_STATION_3_DONE THEN
       "DB8000_PART_STATUS".UNIT_1.STATION_3.PART_A.STATUS.PART_CELL_STATUS_COLOR := 9;
       "DB2401_DBB_DEFINE".PART_STATUS.DBB_1061 := 9;
   END_IF;
   IF #_w2 AND "DB8000_PART_STATUS".UNIT_1.STATION_3.PART_A.STATUS.UNIT_2_STATUS.FACE_N_STATION_4_DONE THEN
       "DB8000_PART_STATUS".UNIT_1.STATION_3.PART_A.STATUS.PART_CELL_STATUS_COLOR := 10;
       "DB2401_DBB_DEFINE".PART_STATUS.DBB_1061 := 10;
   END_IF;
   IF #_w2 AND "DB8000_PART_STATUS".UNIT_1.STATION_3.PART_A.STATUS.CELL_STATUS.U2_ONE_FACE_DONE_ROTATED THEN
       "DB8000_PART_STATUS".UNIT_1.STATION_3.PART_A.STATUS.PART_CELL_STATUS_COLOR := 11;
       "DB2401_DBB_DEFINE".PART_STATUS.DBB_1061 := 11;
   END_IF;
   IF #_w2 AND "DB8000_PART_STATUS".UNIT_1.STATION_3.PART_A.STATUS.UNIT_2_STATUS.FACE_R_STATION_2_DONE THEN
       "DB8000_PART_STATUS".UNIT_1.STATION_3.PART_A.STATUS.PART_CELL_STATUS_COLOR := 12;
       "DB2401_DBB_DEFINE".PART_STATUS.DBB_1061 := 12;
   END_IF;
   IF #_w2 AND "DB8000_PART_STATUS".UNIT_1.STATION_3.PART_A.STATUS.UNIT_2_STATUS.FACE_R_STATION_3_DONE THEN
       "DB8000_PART_STATUS".UNIT_1.STATION_3.PART_A.STATUS.PART_CELL_STATUS_COLOR := 13;
       "DB2401_DBB_DEFINE".PART_STATUS.DBB_1061 := 13;
   END_IF;
   IF #_w2 AND "DB8000_PART_STATUS".UNIT_1.STATION_3.PART_A.STATUS.UNIT_2_STATUS.FACE_R_STATION_4_DONE THEN
       "DB8000_PART_STATUS".UNIT_1.STATION_3.PART_A.STATUS.PART_CELL_STATUS_COLOR := 14;
       "DB2401_DBB_DEFINE".PART_STATUS.DBB_1061 := 14;
   END_IF;
   IF #_w2 AND "DB8000_PART_STATUS".UNIT_1.STATION_3.PART_A.STATUS.CELL_STATUS.U2_DONE_IN_TRANSIT THEN
       "DB8000_PART_STATUS".UNIT_1.STATION_3.PART_A.STATUS.PART_CELL_STATUS_COLOR := 15;
       "DB2401_DBB_DEFINE".PART_STATUS.DBB_1061 := 15;
   END_IF;
   IF #_w2 AND "DB8000_PART_STATUS".UNIT_1.STATION_3.PART_A.STATUS.CELL_STATUS.COOLING_DONE THEN
       "DB8000_PART_STATUS".UNIT_1.STATION_3.PART_A.STATUS.PART_CELL_STATUS_COLOR := 16;
       "DB2401_DBB_DEFINE".PART_STATUS.DBB_1061 := 16;
   END_IF;
   IF #_w2 AND "DB8000_PART_STATUS".UNIT_1.STATION_3.PART_A.STATUS.CELL_STATUS.INSPECTION_DONE THEN
       "DB8000_PART_STATUS".UNIT_1.STATION_3.PART_A.STATUS.PART_CELL_STATUS_COLOR := 17;
       "DB2401_DBB_DEFINE".PART_STATUS.DBB_1061 := 17;
   END_IF;
   IF #_w2 AND "DB8000_PART_STATUS".UNIT_1.STATION_3.PART_A.STATUS.MASTER_PART THEN
       "DB8000_PART_STATUS".UNIT_1.STATION_3.PART_A.STATUS.PART_CELL_STATUS_COLOR := 99;
       "DB2401_DBB_DEFINE".PART_STATUS.DBB_1061 := 99;
   END_IF;
END_REGION

REGION Network 27: PART A STATION 4 COLOR STATUS
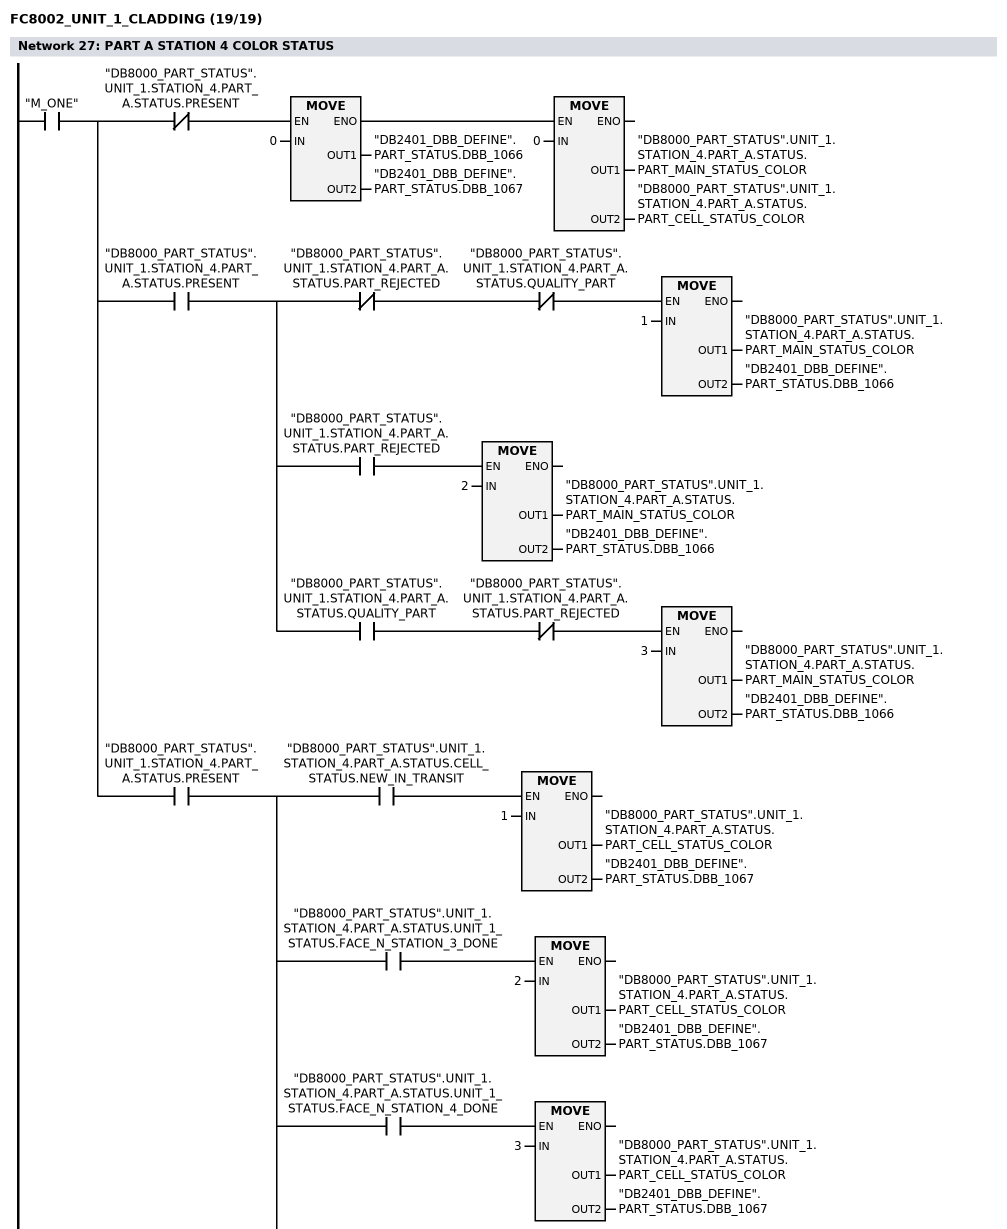
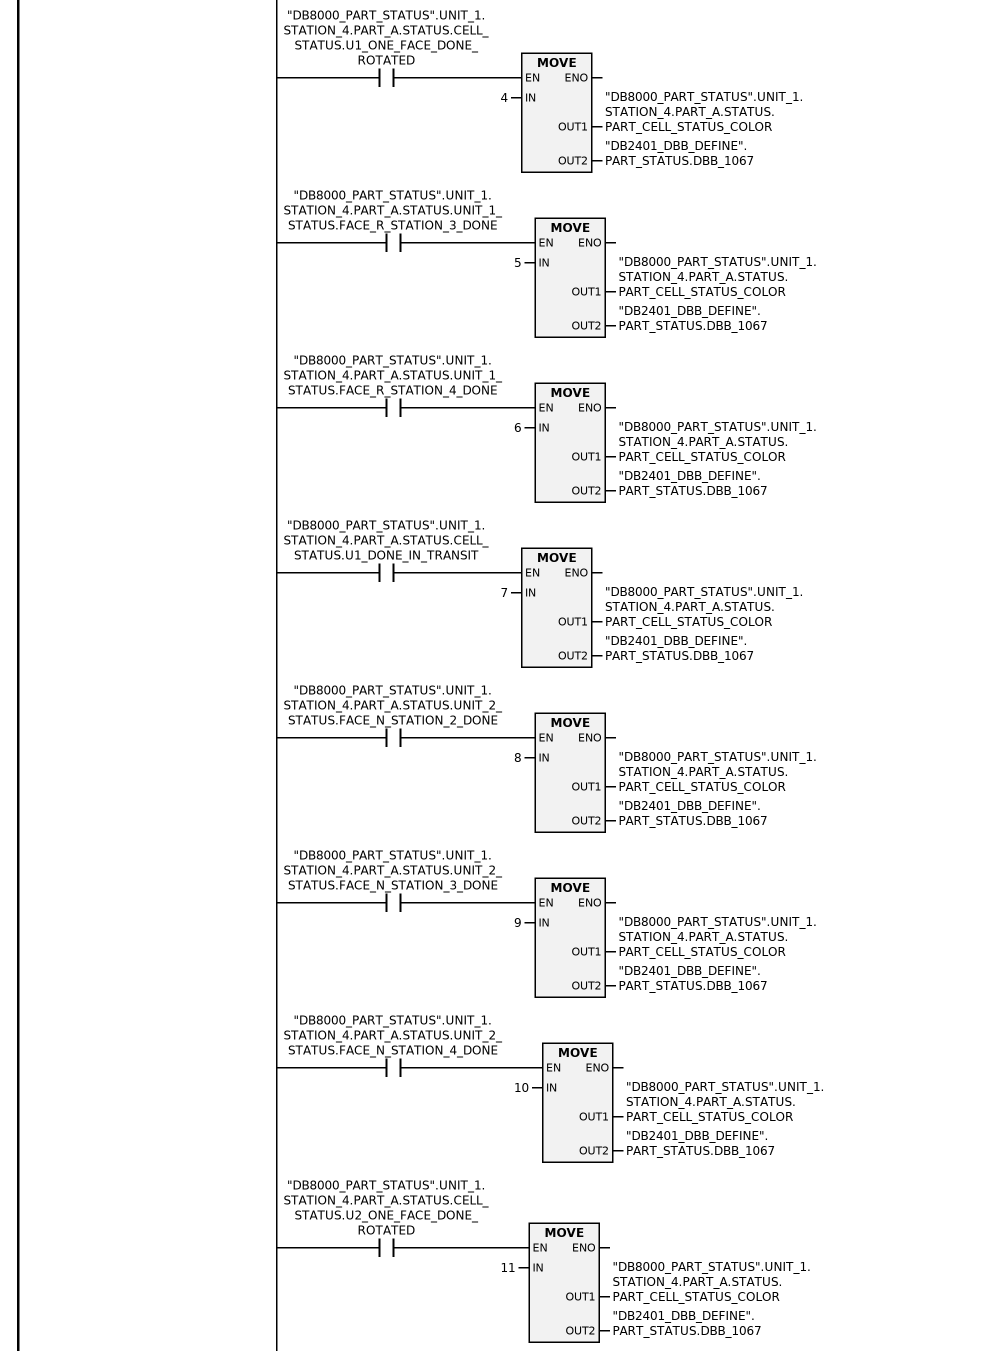
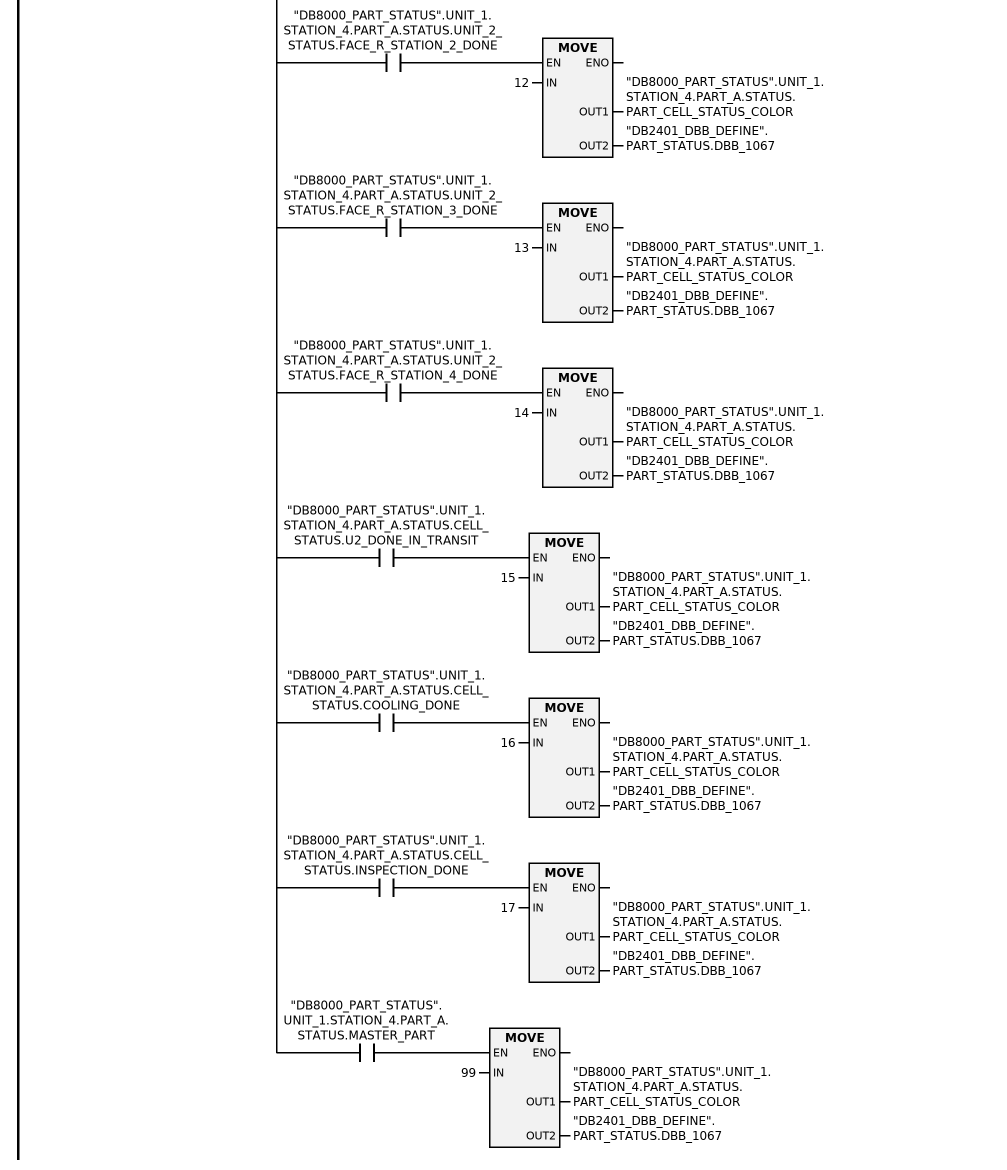
   RUNG wire#powerrail
      Contact( "M_ONE" )
      wire#w1
      I_Contact( "DB8000_PART_STATUS".UNIT_1.STATION_4.PART_A.STATUS.PRESENT )
      { S7_GenerateENO := "TRUE" } Move(in := 0, out1 => "DB2401_DBB_DEFINE".PART_STATUS.DBB_1066, out2 => "DB2401_DBB_DEFINE".PART_STATUS.DBB_1067)
      { S7_GenerateENO := "TRUE" } Move(in := 0, out1 => "DB8000_PART_STATUS".UNIT_1.STATION_4.PART_A.STATUS.PART_MAIN_STATUS_COLOR, out2 => "DB8000_PART_STATUS".UNIT_1.STATION_4.PART_A.STATUS.PART_CELL_STATUS_COLOR)
   END_RUNG
   RUNG wire#w1
      Contact( "DB8000_PART_STATUS".UNIT_1.STATION_4.PART_A.STATUS.PRESENT )
      wire#w2
      I_Contact( "DB8000_PART_STATUS".UNIT_1.STATION_4.PART_A.STATUS.PART_REJECTED )
      I_Contact( "DB8000_PART_STATUS".UNIT_1.STATION_4.PART_A.STATUS.QUALITY_PART )
      { S7_GenerateENO := "TRUE" } Move(in := 1, out1 => "DB8000_PART_STATUS".UNIT_1.STATION_4.PART_A.STATUS.PART_MAIN_STATUS_COLOR, out2 => "DB2401_DBB_DEFINE".PART_STATUS.DBB_1066)
   END_RUNG
   RUNG wire#w2
      Contact( "DB8000_PART_STATUS".UNIT_1.STATION_4.PART_A.STATUS.PART_REJECTED )
      { S7_GenerateENO := "TRUE" } Move(in := 2, out1 => "DB8000_PART_STATUS".UNIT_1.STATION_4.PART_A.STATUS.PART_MAIN_STATUS_COLOR, out2 => "DB2401_DBB_DEFINE".PART_STATUS.DBB_1066)
   END_RUNG
   RUNG wire#w2
      Contact( "DB8000_PART_STATUS".UNIT_1.STATION_4.PART_A.STATUS.QUALITY_PART )
      I_Contact( "DB8000_PART_STATUS".UNIT_1.STATION_4.PART_A.STATUS.PART_REJECTED )
      { S7_GenerateENO := "TRUE" } Move(in := 3, out1 => "DB8000_PART_STATUS".UNIT_1.STATION_4.PART_A.STATUS.PART_MAIN_STATUS_COLOR, out2 => "DB2401_DBB_DEFINE".PART_STATUS.DBB_1066)
   END_RUNG
   RUNG wire#w1
      Contact( "DB8000_PART_STATUS".UNIT_1.STATION_4.PART_A.STATUS.PRESENT )
      wire#w3
      Contact( "DB8000_PART_STATUS".UNIT_1.STATION_4.PART_A.STATUS.CELL_STATUS.NEW_IN_TRANSIT )
      { S7_GenerateENO := "TRUE" } Move(in := 1, out1 => "DB8000_PART_STATUS".UNIT_1.STATION_4.PART_A.STATUS.PART_CELL_STATUS_COLOR, out2 => "DB2401_DBB_DEFINE".PART_STATUS.DBB_1067)
   END_RUNG
   RUNG wire#w3
      Contact( "DB8000_PART_STATUS".UNIT_1.STATION_4.PART_A.STATUS.UNIT_1_STATUS.FACE_N_STATION_3_DONE )
      { S7_GenerateENO := "TRUE" } Move(in := 2, out1 => "DB8000_PART_STATUS".UNIT_1.STATION_4.PART_A.STATUS.PART_CELL_STATUS_COLOR, out2 => "DB2401_DBB_DEFINE".PART_STATUS.DBB_1067)
   END_RUNG
   RUNG wire#w3
      Contact( "DB8000_PART_STATUS".UNIT_1.STATION_4.PART_A.STATUS.UNIT_1_STATUS.FACE_N_STATION_4_DONE )
      { S7_GenerateENO := "TRUE" } Move(in := 3, out1 => "DB8000_PART_STATUS".UNIT_1.STATION_4.PART_A.STATUS.PART_CELL_STATUS_COLOR, out2 => "DB2401_DBB_DEFINE".PART_STATUS.DBB_1067)
   END_RUNG
   RUNG wire#w3
      Contact( "DB8000_PART_STATUS".UNIT_1.STATION_4.PART_A.STATUS.CELL_STATUS.U1_ONE_FACE_DONE_ROTATED )
      { S7_GenerateENO := "TRUE" } Move(in := 4, out1 => "DB8000_PART_STATUS".UNIT_1.STATION_4.PART_A.STATUS.PART_CELL_STATUS_COLOR, out2 => "DB2401_DBB_DEFINE".PART_STATUS.DBB_1067)
   END_RUNG
   RUNG wire#w3
      Contact( "DB8000_PART_STATUS".UNIT_1.STATION_4.PART_A.STATUS.UNIT_1_STATUS.FACE_R_STATION_3_DONE )
      { S7_GenerateENO := "TRUE" } Move(in := 5, out1 => "DB8000_PART_STATUS".UNIT_1.STATION_4.PART_A.STATUS.PART_CELL_STATUS_COLOR, out2 => "DB2401_DBB_DEFINE".PART_STATUS.DBB_1067)
   END_RUNG
   RUNG wire#w3
      Contact( "DB8000_PART_STATUS".UNIT_1.STATION_4.PART_A.STATUS.UNIT_1_STATUS.FACE_R_STATION_4_DONE )
      { S7_GenerateENO := "TRUE" } Move(in := 6, out1 => "DB8000_PART_STATUS".UNIT_1.STATION_4.PART_A.STATUS.PART_CELL_STATUS_COLOR, out2 => "DB2401_DBB_DEFINE".PART_STATUS.DBB_1067)
   END_RUNG
   RUNG wire#w3
      Contact( "DB8000_PART_STATUS".UNIT_1.STATION_4.PART_A.STATUS.CELL_STATUS.U1_DONE_IN_TRANSIT )
      { S7_GenerateENO := "TRUE" } Move(in := 7, out1 => "DB8000_PART_STATUS".UNIT_1.STATION_4.PART_A.STATUS.PART_CELL_STATUS_COLOR, out2 => "DB2401_DBB_DEFINE".PART_STATUS.DBB_1067)
   END_RUNG
   RUNG wire#w3
      Contact( "DB8000_PART_STATUS".UNIT_1.STATION_4.PART_A.STATUS.UNIT_2_STATUS.FACE_N_STATION_2_DONE )
      { S7_GenerateENO := "TRUE" } Move(in := 8, out1 => "DB8000_PART_STATUS".UNIT_1.STATION_4.PART_A.STATUS.PART_CELL_STATUS_COLOR, out2 => "DB2401_DBB_DEFINE".PART_STATUS.DBB_1067)
   END_RUNG
   RUNG wire#w3
      Contact( "DB8000_PART_STATUS".UNIT_1.STATION_4.PART_A.STATUS.UNIT_2_STATUS.FACE_N_STATION_3_DONE )
      Move(in := 9, out1 => "DB8000_PART_STATUS".UNIT_1.STATION_4.PART_A.STATUS.PART_CELL_STATUS_COLOR, out2 => "DB2401_DBB_DEFINE".PART_STATUS.DBB_1067)
   END_RUNG
   RUNG wire#w3
      Contact( "DB8000_PART_STATUS".UNIT_1.STATION_4.PART_A.STATUS.UNIT_2_STATUS.FACE_N_STATION_4_DONE )
      Move(in := 10, out1 => "DB8000_PART_STATUS".UNIT_1.STATION_4.PART_A.STATUS.PART_CELL_STATUS_COLOR, out2 => "DB2401_DBB_DEFINE".PART_STATUS.DBB_1067)
   END_RUNG
   RUNG wire#w3
      Contact( "DB8000_PART_STATUS".UNIT_1.STATION_4.PART_A.STATUS.CELL_STATUS.U2_ONE_FACE_DONE_ROTATED )
      Move(in := 11, out1 => "DB8000_PART_STATUS".UNIT_1.STATION_4.PART_A.STATUS.PART_CELL_STATUS_COLOR, out2 => "DB2401_DBB_DEFINE".PART_STATUS.DBB_1067)
   END_RUNG
   RUNG wire#w3
      Contact( "DB8000_PART_STATUS".UNIT_1.STATION_4.PART_A.STATUS.UNIT_2_STATUS.FACE_R_STATION_2_DONE )
      Move(in := 12, out1 => "DB8000_PART_STATUS".UNIT_1.STATION_4.PART_A.STATUS.PART_CELL_STATUS_COLOR, out2 => "DB2401_DBB_DEFINE".PART_STATUS.DBB_1067)
   END_RUNG
   RUNG wire#w3
      Contact( "DB8000_PART_STATUS".UNIT_1.STATION_4.PART_A.STATUS.UNIT_2_STATUS.FACE_R_STATION_3_DONE )
      Move(in := 13, out1 => "DB8000_PART_STATUS".UNIT_1.STATION_4.PART_A.STATUS.PART_CELL_STATUS_COLOR, out2 => "DB2401_DBB_DEFINE".PART_STATUS.DBB_1067)
   END_RUNG
   RUNG wire#w3
      Contact( "DB8000_PART_STATUS".UNIT_1.STATION_4.PART_A.STATUS.UNIT_2_STATUS.FACE_R_STATION_4_DONE )
      Move(in := 14, out1 => "DB8000_PART_STATUS".UNIT_1.STATION_4.PART_A.STATUS.PART_CELL_STATUS_COLOR, out2 => "DB2401_DBB_DEFINE".PART_STATUS.DBB_1067)
   END_RUNG
   RUNG wire#w3
      Contact( "DB8000_PART_STATUS".UNIT_1.STATION_4.PART_A.STATUS.CELL_STATUS.U2_DONE_IN_TRANSIT )
      Move(in := 15, out1 => "DB8000_PART_STATUS".UNIT_1.STATION_4.PART_A.STATUS.PART_CELL_STATUS_COLOR, out2 => "DB2401_DBB_DEFINE".PART_STATUS.DBB_1067)
   END_RUNG
   RUNG wire#w3
      Contact( "DB8000_PART_STATUS".UNIT_1.STATION_4.PART_A.STATUS.CELL_STATUS.COOLING_DONE )
      Move(in := 16, out1 => "DB8000_PART_STATUS".UNIT_1.STATION_4.PART_A.STATUS.PART_CELL_STATUS_COLOR, out2 => "DB2401_DBB_DEFINE".PART_STATUS.DBB_1067)
   END_RUNG
   RUNG wire#w3
      Contact( "DB8000_PART_STATUS".UNIT_1.STATION_4.PART_A.STATUS.CELL_STATUS.INSPECTION_DONE )
      Move(in := 17, out1 => "DB8000_PART_STATUS".UNIT_1.STATION_4.PART_A.STATUS.PART_CELL_STATUS_COLOR, out2 => "DB2401_DBB_DEFINE".PART_STATUS.DBB_1067)
   END_RUNG
   RUNG wire#w3
      Contact( "DB8000_PART_STATUS".UNIT_1.STATION_4.PART_A.STATUS.MASTER_PART )
      Move(in := 99, out1 => "DB8000_PART_STATUS".UNIT_1.STATION_4.PART_A.STATUS.PART_CELL_STATUS_COLOR, out2 => "DB2401_DBB_DEFINE".PART_STATUS.DBB_1067)
   END_RUNG
   // the same network as SCL:
   // ENO of a box is taken as its EN; it also drops when the box reports an error
   IF "M_ONE" AND NOT "DB8000_PART_STATUS".UNIT_1.STATION_4.PART_A.STATUS.PRESENT THEN
       "DB2401_DBB_DEFINE".PART_STATUS.DBB_1066 := 0;
       "DB2401_DBB_DEFINE".PART_STATUS.DBB_1067 := 0;
       "DB8000_PART_STATUS".UNIT_1.STATION_4.PART_A.STATUS.PART_MAIN_STATUS_COLOR := 0;
       "DB8000_PART_STATUS".UNIT_1.STATION_4.PART_A.STATUS.PART_CELL_STATUS_COLOR := 0;
   END_IF;
   #_w1 := "M_ONE" AND "DB8000_PART_STATUS".UNIT_1.STATION_4.PART_A.STATUS.PRESENT;
   IF #_w1 AND NOT "DB8000_PART_STATUS".UNIT_1.STATION_4.PART_A.STATUS.PART_REJECTED AND NOT "DB8000_PART_STATUS".UNIT_1.STATION_4.PART_A.STATUS.QUALITY_PART THEN
       "DB8000_PART_STATUS".UNIT_1.STATION_4.PART_A.STATUS.PART_MAIN_STATUS_COLOR := 1;
       "DB2401_DBB_DEFINE".PART_STATUS.DBB_1066 := 1;
   END_IF;
   IF #_w1 AND "DB8000_PART_STATUS".UNIT_1.STATION_4.PART_A.STATUS.PART_REJECTED THEN
       "DB8000_PART_STATUS".UNIT_1.STATION_4.PART_A.STATUS.PART_MAIN_STATUS_COLOR := 2;
       "DB2401_DBB_DEFINE".PART_STATUS.DBB_1066 := 2;
   END_IF;
   IF #_w1 AND "DB8000_PART_STATUS".UNIT_1.STATION_4.PART_A.STATUS.QUALITY_PART AND NOT "DB8000_PART_STATUS".UNIT_1.STATION_4.PART_A.STATUS.PART_REJECTED THEN
       "DB8000_PART_STATUS".UNIT_1.STATION_4.PART_A.STATUS.PART_MAIN_STATUS_COLOR := 3;
       "DB2401_DBB_DEFINE".PART_STATUS.DBB_1066 := 3;
   END_IF;
   #_w2 := "M_ONE" AND "DB8000_PART_STATUS".UNIT_1.STATION_4.PART_A.STATUS.PRESENT;
   IF #_w2 AND "DB8000_PART_STATUS".UNIT_1.STATION_4.PART_A.STATUS.CELL_STATUS.NEW_IN_TRANSIT THEN
       "DB8000_PART_STATUS".UNIT_1.STATION_4.PART_A.STATUS.PART_CELL_STATUS_COLOR := 1;
       "DB2401_DBB_DEFINE".PART_STATUS.DBB_1067 := 1;
   END_IF;
   IF #_w2 AND "DB8000_PART_STATUS".UNIT_1.STATION_4.PART_A.STATUS.UNIT_1_STATUS.FACE_N_STATION_3_DONE THEN
       "DB8000_PART_STATUS".UNIT_1.STATION_4.PART_A.STATUS.PART_CELL_STATUS_COLOR := 2;
       "DB2401_DBB_DEFINE".PART_STATUS.DBB_1067 := 2;
   END_IF;
   IF #_w2 AND "DB8000_PART_STATUS".UNIT_1.STATION_4.PART_A.STATUS.UNIT_1_STATUS.FACE_N_STATION_4_DONE THEN
       "DB8000_PART_STATUS".UNIT_1.STATION_4.PART_A.STATUS.PART_CELL_STATUS_COLOR := 3;
       "DB2401_DBB_DEFINE".PART_STATUS.DBB_1067 := 3;
   END_IF;
   IF #_w2 AND "DB8000_PART_STATUS".UNIT_1.STATION_4.PART_A.STATUS.CELL_STATUS.U1_ONE_FACE_DONE_ROTATED THEN
       "DB8000_PART_STATUS".UNIT_1.STATION_4.PART_A.STATUS.PART_CELL_STATUS_COLOR := 4;
       "DB2401_DBB_DEFINE".PART_STATUS.DBB_1067 := 4;
   END_IF;
   IF #_w2 AND "DB8000_PART_STATUS".UNIT_1.STATION_4.PART_A.STATUS.UNIT_1_STATUS.FACE_R_STATION_3_DONE THEN
       "DB8000_PART_STATUS".UNIT_1.STATION_4.PART_A.STATUS.PART_CELL_STATUS_COLOR := 5;
       "DB2401_DBB_DEFINE".PART_STATUS.DBB_1067 := 5;
   END_IF;
   IF #_w2 AND "DB8000_PART_STATUS".UNIT_1.STATION_4.PART_A.STATUS.UNIT_1_STATUS.FACE_R_STATION_4_DONE THEN
       "DB8000_PART_STATUS".UNIT_1.STATION_4.PART_A.STATUS.PART_CELL_STATUS_COLOR := 6;
       "DB2401_DBB_DEFINE".PART_STATUS.DBB_1067 := 6;
   END_IF;
   IF #_w2 AND "DB8000_PART_STATUS".UNIT_1.STATION_4.PART_A.STATUS.CELL_STATUS.U1_DONE_IN_TRANSIT THEN
       "DB8000_PART_STATUS".UNIT_1.STATION_4.PART_A.STATUS.PART_CELL_STATUS_COLOR := 7;
       "DB2401_DBB_DEFINE".PART_STATUS.DBB_1067 := 7;
   END_IF;
   IF #_w2 AND "DB8000_PART_STATUS".UNIT_1.STATION_4.PART_A.STATUS.UNIT_2_STATUS.FACE_N_STATION_2_DONE THEN
       "DB8000_PART_STATUS".UNIT_1.STATION_4.PART_A.STATUS.PART_CELL_STATUS_COLOR := 8;
       "DB2401_DBB_DEFINE".PART_STATUS.DBB_1067 := 8;
   END_IF;
   IF #_w2 AND "DB8000_PART_STATUS".UNIT_1.STATION_4.PART_A.STATUS.UNIT_2_STATUS.FACE_N_STATION_3_DONE THEN
       "DB8000_PART_STATUS".UNIT_1.STATION_4.PART_A.STATUS.PART_CELL_STATUS_COLOR := 9;
       "DB2401_DBB_DEFINE".PART_STATUS.DBB_1067 := 9;
   END_IF;
   IF #_w2 AND "DB8000_PART_STATUS".UNIT_1.STATION_4.PART_A.STATUS.UNIT_2_STATUS.FACE_N_STATION_4_DONE THEN
       "DB8000_PART_STATUS".UNIT_1.STATION_4.PART_A.STATUS.PART_CELL_STATUS_COLOR := 10;
       "DB2401_DBB_DEFINE".PART_STATUS.DBB_1067 := 10;
   END_IF;
   IF #_w2 AND "DB8000_PART_STATUS".UNIT_1.STATION_4.PART_A.STATUS.CELL_STATUS.U2_ONE_FACE_DONE_ROTATED THEN
       "DB8000_PART_STATUS".UNIT_1.STATION_4.PART_A.STATUS.PART_CELL_STATUS_COLOR := 11;
       "DB2401_DBB_DEFINE".PART_STATUS.DBB_1067 := 11;
   END_IF;
   IF #_w2 AND "DB8000_PART_STATUS".UNIT_1.STATION_4.PART_A.STATUS.UNIT_2_STATUS.FACE_R_STATION_2_DONE THEN
       "DB8000_PART_STATUS".UNIT_1.STATION_4.PART_A.STATUS.PART_CELL_STATUS_COLOR := 12;
       "DB2401_DBB_DEFINE".PART_STATUS.DBB_1067 := 12;
   END_IF;
   IF #_w2 AND "DB8000_PART_STATUS".UNIT_1.STATION_4.PART_A.STATUS.UNIT_2_STATUS.FACE_R_STATION_3_DONE THEN
       "DB8000_PART_STATUS".UNIT_1.STATION_4.PART_A.STATUS.PART_CELL_STATUS_COLOR := 13;
       "DB2401_DBB_DEFINE".PART_STATUS.DBB_1067 := 13;
   END_IF;
   IF #_w2 AND "DB8000_PART_STATUS".UNIT_1.STATION_4.PART_A.STATUS.UNIT_2_STATUS.FACE_R_STATION_4_DONE THEN
       "DB8000_PART_STATUS".UNIT_1.STATION_4.PART_A.STATUS.PART_CELL_STATUS_COLOR := 14;
       "DB2401_DBB_DEFINE".PART_STATUS.DBB_1067 := 14;
   END_IF;
   IF #_w2 AND "DB8000_PART_STATUS".UNIT_1.STATION_4.PART_A.STATUS.CELL_STATUS.U2_DONE_IN_TRANSIT THEN
       "DB8000_PART_STATUS".UNIT_1.STATION_4.PART_A.STATUS.PART_CELL_STATUS_COLOR := 15;
       "DB2401_DBB_DEFINE".PART_STATUS.DBB_1067 := 15;
   END_IF;
   IF #_w2 AND "DB8000_PART_STATUS".UNIT_1.STATION_4.PART_A.STATUS.CELL_STATUS.COOLING_DONE THEN
       "DB8000_PART_STATUS".UNIT_1.STATION_4.PART_A.STATUS.PART_CELL_STATUS_COLOR := 16;
       "DB2401_DBB_DEFINE".PART_STATUS.DBB_1067 := 16;
   END_IF;
   IF #_w2 AND "DB8000_PART_STATUS".UNIT_1.STATION_4.PART_A.STATUS.CELL_STATUS.INSPECTION_DONE THEN
       "DB8000_PART_STATUS".UNIT_1.STATION_4.PART_A.STATUS.PART_CELL_STATUS_COLOR := 17;
       "DB2401_DBB_DEFINE".PART_STATUS.DBB_1067 := 17;
   END_IF;
   IF #_w2 AND "DB8000_PART_STATUS".UNIT_1.STATION_4.PART_A.STATUS.MASTER_PART THEN
       "DB8000_PART_STATUS".UNIT_1.STATION_4.PART_A.STATUS.PART_CELL_STATUS_COLOR := 99;
       "DB2401_DBB_DEFINE".PART_STATUS.DBB_1067 := 99;
   END_IF;
END_REGION
END_FUNCTION
